TYPE st_NeedleChageBoxData :
STRUCT
	//圓帶位置
	AllocationNo 	:INT;
	//倉儲儲位
	StorageInfor	:INT;
	//盒子順序
	BoxOrder 		:INT;
END_STRUCT
END_TYPE

(* stored: Version 1.1.0.1, ProductVersion 3.1.4024.13
   DUT st_NeedleChageBoxData: Id {a9c060ed-fd3b-41d7-8e20-05ea24a110b9} *)
